// SIMATIC STEP 7 (V5.x) project LOCO#1ON_BOARD_PLC(TATA)
// CPU: CPU 315-2 DP
// station: P_ADR_BUS
// station: Hardware
// station: OB_PLC_QL--1
// program: S7 Program(1)

SYMBOL_TABLE
"RDREC"	SFB 52	SFB 52	// Read a Process Data Record
"WRREC"	SFB 53	SFB 53	// Write a Process Data Record
"RD_SINFO"	SFC 6	SFC 6	// Read OB Start Information
"BLKMOV"	SFC 20	SFC 20	// Copy Variables
"FILL"	SFC 21	SFC 21	// Initialize a Memory Area
"RDSYSST"	SFC 51	SFC 51	// Read a System Status List or Partial List
"WR_REC"	SFC 58	SFC 58	// Write Data Record
"RD_REC"	SFC 59	SFC 59	// Read a Data Record
END_SYMBOL_TABLE

// FB 7: know-how protected block, not included

// FB 8: know-how protected block, not included

// FC 1: know-how protected block, not included

// FC 2: know-how protected block, not included

// FC 3: know-how protected block, not included

// FC 4: know-how protected block, not included

FUNCTION FC 10 : VOID
VERSION : 0.1
BEGIN
// (block stored without names or comments; labels and parameter names are numbered)
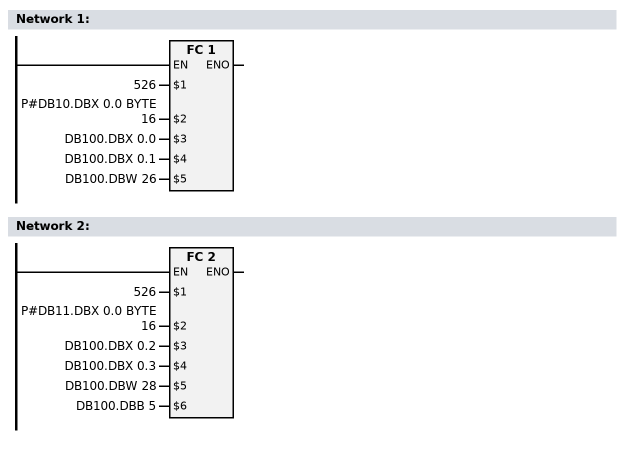
NETWORK
TITLE =
      CALL  FC 1 (
           $1                       := 526,
           $2                       := P#DB10.DBX 0.0 BYTE 16,
           $3                       := DB100.DBX 0.0,
           $4                       := DB100.DBX 0.1,
           $5                       := DB100.DBW 26);
      NOP   0;
NETWORK
TITLE =
      CALL  FC 2 (
           $1                       := 526,
           $2                       := P#DB11.DBX 0.0 BYTE 16,
           $3                       := DB100.DBX 0.2,
           $4                       := DB100.DBX 0.3,
           $5                       := DB100.DBW 28,
           $6                       := DB100.DBB 5);
      NOP   0;
END_FUNCTION

FUNCTION FC 14 : VOID
VERSION : 0.1
BEGIN
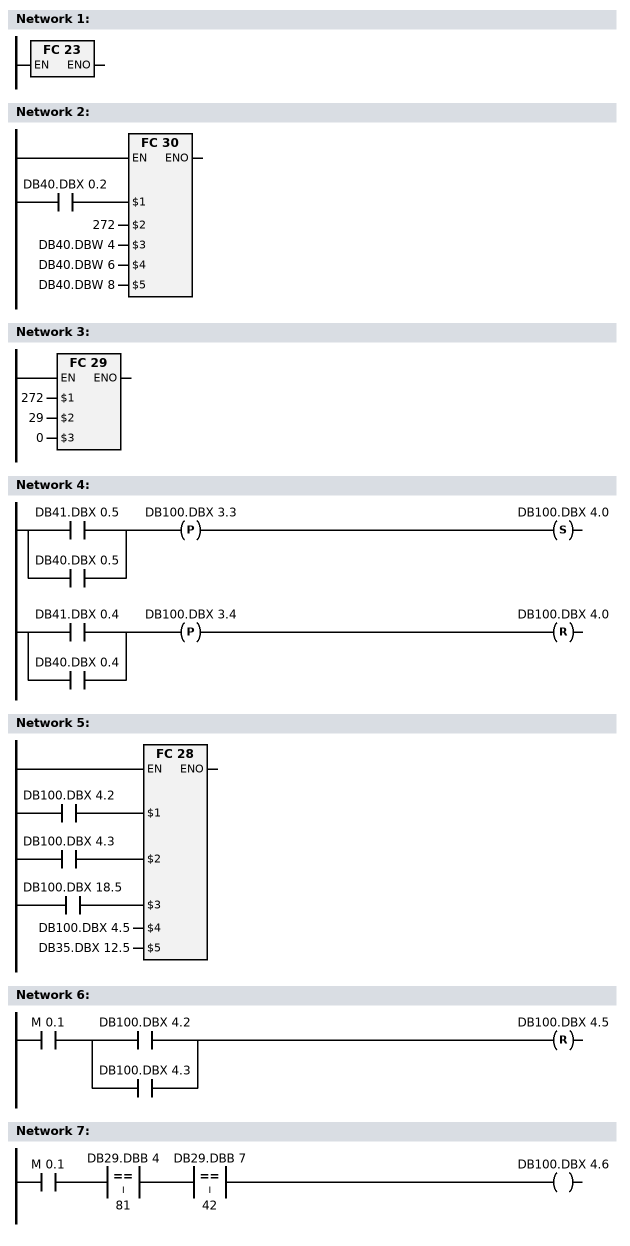
NETWORK
TITLE =
      CALL  FC 23;
      NOP   0;
NETWORK
TITLE =
      A     DB40.DBX 0.2;
      =     L 0.0;
      BLD   103;
      CALL  FC 30 (
           $1                       := L 0.0,
           $2                       := 272,
           $3                       := DB40.DBW 4,
           $4                       := DB40.DBW 6,
           $5                       := DB40.DBW 8);
      NOP   0;
NETWORK
TITLE =
      CALL  FC 29 (
           $1                       := 272,
           $2                       := 29,
           $3                       := 0);
      NOP   0;
NETWORK
TITLE =
      A(;
      O     DB41.DBX 0.5;
      O     DB40.DBX 0.5;
      );
      FP    DB100.DBX 3.3;
      S     DB100.DBX 4.0;
      A(;
      O     DB41.DBX 0.4;
      O     DB40.DBX 0.4;
      );
      FP    DB100.DBX 3.4;
      R     DB100.DBX 4.0;
      NOP   0;
NETWORK
TITLE =
      A     DB100.DBX 4.2;
      =     L 0.0;
      BLD   103;
      A     DB100.DBX 4.3;
      =     L 0.1;
      BLD   103;
      A     DB100.DBX 18.5;
      =     L 0.2;
      BLD   103;
      CALL  FC 28 (
           $1                       := L 0.0,
           $2                       := L 0.1,
           $3                       := L 0.2,
           $4                       := DB100.DBX 4.5,
           $5                       := DB35.DBX 12.5);
      NOP   0;
NETWORK
TITLE =
      A     M 0.1;
      A(;
      O     DB100.DBX 4.2;
      O     DB100.DBX 4.3;
      );
      R     DB100.DBX 4.5;
NETWORK
TITLE =
      A     M 0.1;
      A(;
      L     DB29.DBB 4;
      L     81;
      ==I;
      );
      A(;
      L     DB29.DBB 7;
      L     42;
      ==I;
      );
      =     DB100.DBX 4.6;
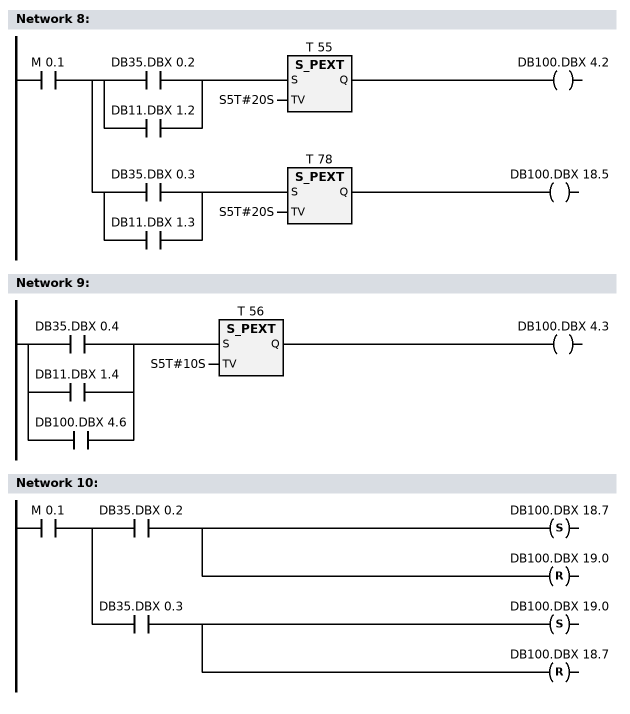
NETWORK
TITLE =
      A     M 0.1;
      =     L 0.0;
      A     L 0.0;
      A(;
      O     DB35.DBX 0.2;
      O     DB11.DBX 1.2;
      );
      L     S5T#20S;
      SE    T 55;
      NOP   0;
      NOP   0;
      NOP   0;
      A     T 55;
      =     DB100.DBX 4.2;
      A     L 0.0;
      A(;
      O     DB35.DBX 0.3;
      O     DB11.DBX 1.3;
      );
      L     S5T#20S;
      SE    T 78;
      NOP   0;
      NOP   0;
      NOP   0;
      A     T 78;
      =     DB100.DBX 18.5;
NETWORK
TITLE =
      A(;
      O     DB35.DBX 0.4;
      O     DB11.DBX 1.4;
      O     DB100.DBX 4.6;
      );
      L     S5T#10S;
      SE    T 56;
      NOP   0;
      NOP   0;
      NOP   0;
      A     T 56;
      =     DB100.DBX 4.3;
NETWORK
TITLE =
      A     M 0.1;
      =     L 0.0;
      A     L 0.0;
      A     DB35.DBX 0.2;
      S     DB100.DBX 18.7;
      R     DB100.DBX 19.0;
      A     L 0.0;
      A     DB35.DBX 0.3;
      S     DB100.DBX 19.0;
      R     DB100.DBX 18.7;
END_FUNCTION

FUNCTION FC 16 : VOID
VERSION : 0.1
BEGIN
// (block stored without names or comments; labels and parameter names are numbered)
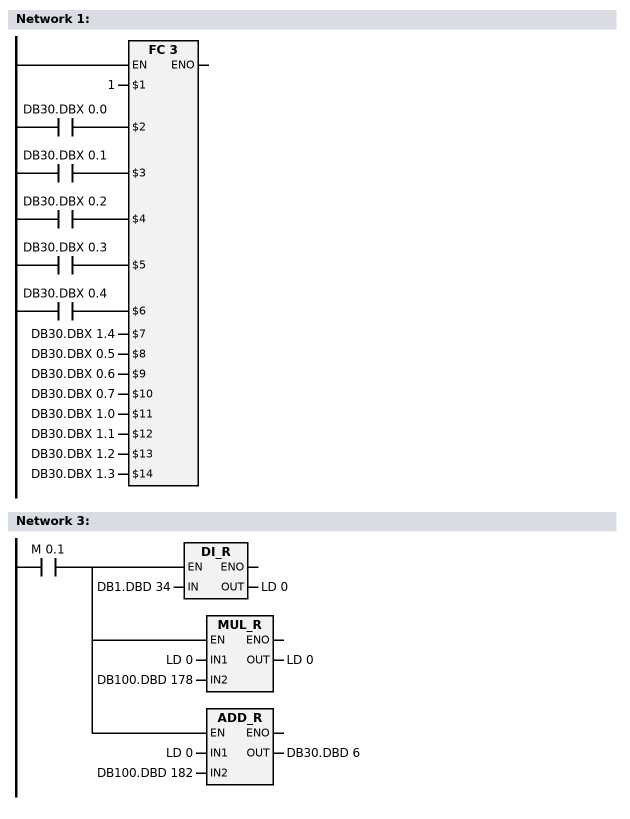
NETWORK
TITLE =
      A     DB30.DBX 0.0;
      =     L 4.0;
      BLD   103;
      A     DB30.DBX 0.1;
      =     L 4.1;
      BLD   103;
      A     DB30.DBX 0.2;
      =     L 4.2;
      BLD   103;
      A     DB30.DBX 0.3;
      =     L 4.3;
      BLD   103;
      A     DB30.DBX 0.4;
      =     L 4.4;
      BLD   103;
      CALL  FC 3 (
           $1                       := 1,
           $2                       := L 4.0,
           $3                       := L 4.1,
           $4                       := L 4.2,
           $5                       := L 4.3,
           $6                       := L 4.4,
           $7                       := DB30.DBX 1.4,
           $8                       := DB30.DBX 0.5,
           $9                       := DB30.DBX 0.6,
           $10                      := DB30.DBX 0.7,
           $11                      := DB30.DBX 1.0,
           $12                      := DB30.DBX 1.1,
           $13                      := DB30.DBX 1.2,
           $14                      := DB30.DBX 1.3);
      NOP   0;
NETWORK
TITLE =
NETWORK
TITLE =
      A     M 0.1;
      =     L 4.0;
      A     L 4.0;
      JNB   M001;
      L     DB1.DBD 34;
      DTR;
      T     LD 0;
M001: NOP   0;
      A     L 4.0;
      JNB   M002;
      L     LD 0;
      L     DB100.DBD 178;
      *R;
      T     LD 0;
M002: NOP   0;
      A     L 4.0;
      JNB   M003;
      L     LD 0;
      L     DB100.DBD 182;
      +R;
      T     DB30.DBD 6;
M003: NOP   0;
END_FUNCTION

FUNCTION FC 19 : VOID
VERSION : 0.1
BEGIN
// (block stored without names or comments; labels and parameter names are numbered)
NETWORK
TITLE =
      A     DB100.DBX 0.4;
      =     L 0.0;
      BLD   103;
      CALL  FC 31 (
           $1                       := L 0.0,
           $2                       := 288,
           $3                       := DB100.DBW 112,
           $4                       := P#M 45.0,
           $5                       := P#M 47.0,
           $6                       := DB31.DBX 2.0,
           $7                       := DB31.DBX 2.1,
           $8                       := DB31.DBX 2.2,
           $9                       := DB31.DBX 6.0,
           $10                      := DB31.DBX 2.3);
      NOP   0;
NETWORK
TITLE =
      L     MW 45;
      T     DB31.DBW 0;
      L     MW 47;
      T     DB31.DBW 4;
END_FUNCTION

FUNCTION FC 20 : VOID
VERSION : 0.1
BEGIN
// (block stored without names or comments; labels and parameter names are numbered)
NETWORK
TITLE =
      A     M 0.1;
      A(;
      L     DB21.DBW 46;
      L     1;
      ==I;
      );
      A(;
      L     DB21.DBB 50;
      L     'P';
      ==I;
      );
      JNB   M001;
      L     DB21.DBW 24;
      T     DB35.DBW 278;
M001: NOP   0;
NETWORK
TITLE =
      A     M 0.1;
      A(;
      L     DB21.DBW 46;
      L     1;
      ==I;
      );
      A(;
      L     DB21.DBB 50;
      L     'C';
      ==I;
      );
      A(;
      L     DB21.DBW 74;
      L     2;
      ==I;
      );
      A(;
      L     DB21.DBB 78;
      L     'P';
      ==I;
      );
      JNB   M002;
      L     DB21.DBW 52;
      T     DB35.DBW 278;
M002: NOP   0;
NETWORK
TITLE =
      A     M 0.1;
      A(;
      L     DB21.DBW 46;
      L     1;
      ==I;
      );
      A(;
      L     DB21.DBB 50;
      L     'C';
      ==I;
      );
      A(;
      L     DB21.DBW 74;
      L     2;
      ==I;
      );
      A(;
      L     DB21.DBB 78;
      L     'C';
      ==I;
      );
      A(;
      L     DB21.DBW 102;
      L     3;
      ==I;
      );
      A(;
      L     DB21.DBB 106;
      L     'P';
      ==I;
      );
      JNB   M003;
      L     DB21.DBW 80;
      T     DB35.DBW 278;
M003: NOP   0;
NETWORK
TITLE =
      A     M 0.1;
      A(;
      L     DB21.DBW 46;
      L     1;
      ==I;
      );
      A(;
      L     DB21.DBB 50;
      L     'C';
      ==I;
      );
      A(;
      L     DB21.DBW 74;
      L     2;
      ==I;
      );
      A(;
      L     DB21.DBB 78;
      L     'C';
      ==I;
      );
      A(;
      L     DB21.DBW 102;
      L     3;
      ==I;
      );
      A(;
      L     DB21.DBB 106;
      L     'C';
      ==I;
      );
      A(;
      L     DB21.DBW 130;
      L     4;
      ==I;
      );
      A(;
      L     DB21.DBB 134;
      L     'P';
      ==I;
      );
      JNB   M004;
      L     DB21.DBW 108;
      T     DB35.DBW 278;
M004: NOP   0;
NETWORK
TITLE =
      A     M 0.1;
      A(;
      L     DB21.DBW 46;
      L     1;
      ==I;
      );
      A(;
      L     DB21.DBB 50;
      L     'C';
      ==I;
      );
      =     L 0.0;
      A     L 0.0;
      JNB   M005;
      L     DB21.DBW 24;
      T     DB35.DBW 280;
M005: NOP   0;
      A     L 0.0;
      JNB   M006;
      L     DB21.DBB 50;
      T     DB35.DBB 284;
M006: NOP   0;
END_FUNCTION

FUNCTION FC 21 : VOID
VERSION : 0.1
BEGIN
// (block stored without names or comments; labels and parameter names are numbered)
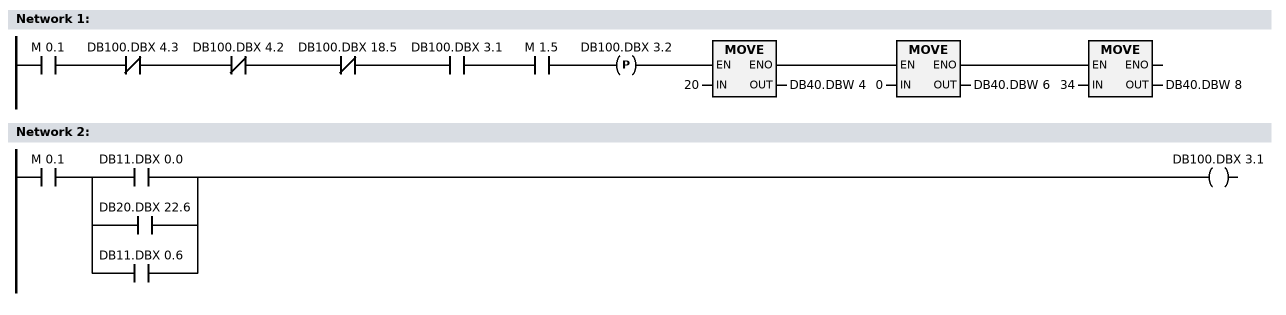
NETWORK
TITLE =
      A(;
      A(;
      A     M 0.1;
      AN    DB100.DBX 4.3;
      AN    DB100.DBX 4.2;
      AN    DB100.DBX 18.5;
      A     DB100.DBX 3.1;
      A     M 1.5;
      FP    DB100.DBX 3.2;
      JNB   M001;
      L     20;
      T     DB40.DBW 4;
      SET;
      SAVE;
      CLR;
M001: A     BR;
      );
      JNB   M002;
      L     0;
      T     DB40.DBW 6;
      SET;
      SAVE;
      CLR;
M002: A     BR;
      );
      JNB   M003;
      L     34;
      T     DB40.DBW 8;
M003: NOP   0;
NETWORK
TITLE =
      A     M 0.1;
      A(;
      O     DB11.DBX 0.0;
      O     DB20.DBX 22.6;
      O     DB11.DBX 0.6;
      );
      =     DB100.DBX 3.1;
END_FUNCTION

FUNCTION FC 22 : VOID
VERSION : 0.1
BEGIN
// (block stored without names or comments; labels and parameter names are numbered)
NETWORK
TITLE =
      A     DB41.DBX 0.4;
      A(;
      L     DB29.DBB 8;
      L     B#16#3;
      ==I;
      );
      A(;
      L     DB29.DBB 11;
      L     32;
      ==I;
      );
      =     DB100.DBX 15.1;
      A     DB100.DBX 15.1;
      FP    DB100.DBX 15.7;
      JNB   M001;
      CALL  "FILL" (
           BVAL                     := P#DB29.DBX 0.0 BYTE 30,
           RET_VAL                  := DB100.DBW 122,
           BLK                      := P#DB17.DBX 0.0 BYTE 30);
M001: NOP   0;
NETWORK
TITLE =
      A     DB41.DBX 0.4;
      A(;
      L     DB29.DBB 8;
      L     B#16#2;
      ==I;
      );
      A(;
      L     DB29.DBB 11;
      L     38;
      ==I;
      );
      =     DB100.DBX 15.0;
      A     DB100.DBX 15.0;
      FP    DB100.DBX 15.5;
      JNB   M002;
      CALL  "FILL" (
           BVAL                     := P#DB29.DBX 0.0 BYTE 34,
           RET_VAL                  := DB100.DBW 120,
           BLK                      := P#DB19.DBX 0.0 BYTE 34);
M002: NOP   0;
NETWORK
TITLE =
      A     DB41.DBX 0.4;
      A(;
      L     DB29.DBB 8;
      L     B#16#4;
      ==I;
      );
      A(;
      L     DB29.DBB 11;
      L     30;
      ==I;
      );
      =     DB100.DBX 15.2;
      A     DB100.DBX 15.2;
      FP    DB100.DBX 15.6;
      JNB   M003;
      CALL  "FILL" (
           BVAL                     := P#DB29.DBX 0.0 BYTE 30,
           RET_VAL                  := DB100.DBW 124,
           BLK                      := P#DB18.DBX 0.0 BYTE 30);
M003: NOP   0;
NETWORK
TITLE =
      A     DB41.DBX 0.4;
      A(;
      L     DB29.DBB 8;
      L     B#16#10;
      ==I;
      );
      A(;
      L     DB29.DBB 11;
      L     167;
      ==I;
      );
      =     DB100.DBX 15.4;
      A     DB100.DBX 15.4;
      FP    DB100.DBX 16.0;
      JNB   M004;
      CALL  "FILL" (
           BVAL                     := P#DB29.DBX 0.0 BYTE 167,
           RET_VAL                  := DB100.DBW 128,
           BLK                      := P#DB21.DBX 0.0 BYTE 167);
M004: NOP   0;
END_FUNCTION

FUNCTION FC 23 : VOID
VERSION : 0.1
BEGIN
// (block stored without names or comments; labels and parameter names are numbered)
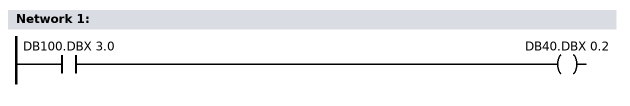
NETWORK
TITLE =
      A     DB100.DBX 3.0;
      =     DB40.DBX 0.2;
END_FUNCTION

FUNCTION FC 24 : VOID
VERSION : 0.1
BEGIN
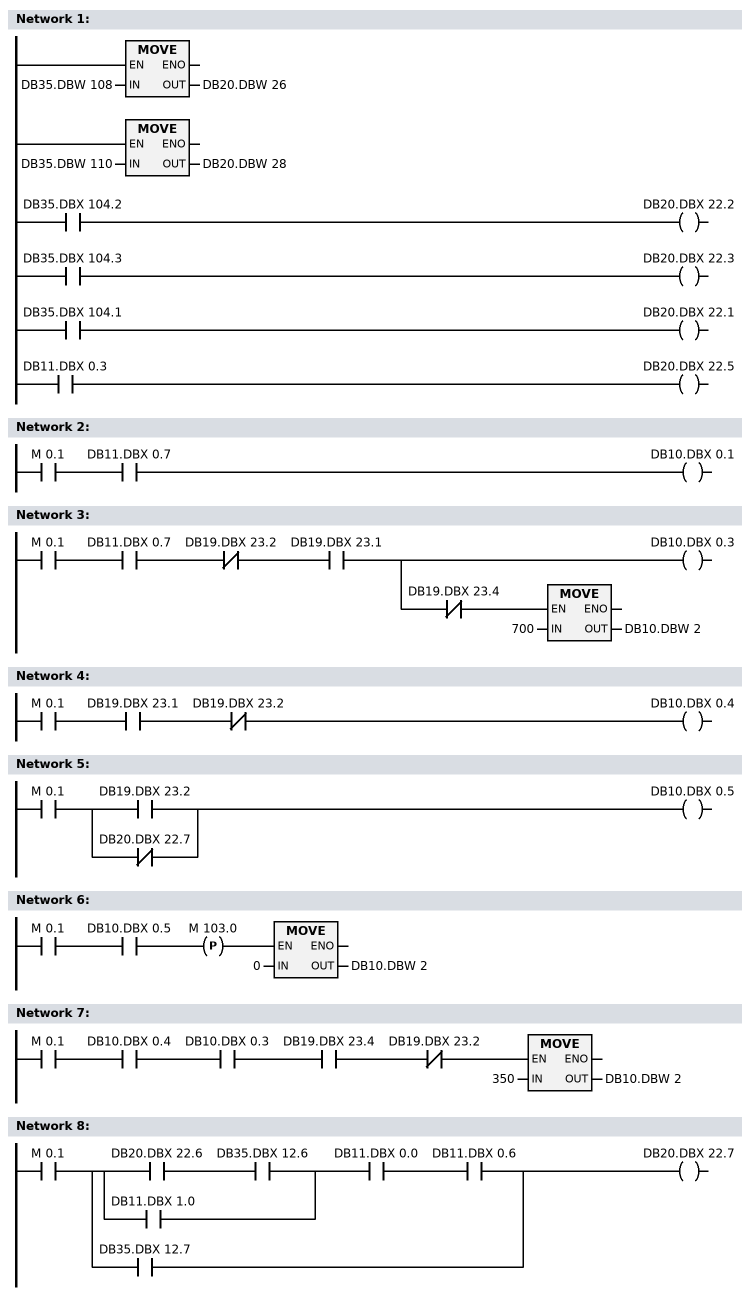
NETWORK
TITLE =
      L     DB35.DBW 108;
      T     DB20.DBW 26;
      L     DB35.DBW 110;
      T     DB20.DBW 28;
      A     DB35.DBX 104.2;
      =     DB20.DBX 22.2;
      A     DB35.DBX 104.3;
      =     DB20.DBX 22.3;
      A     DB35.DBX 104.1;
      =     DB20.DBX 22.1;
      A     DB11.DBX 0.3;
      =     DB20.DBX 22.5;
NETWORK
TITLE =
      A     M 0.1;
      A     DB11.DBX 0.7;
      =     DB10.DBX 0.1;
NETWORK
TITLE =
      A     M 0.1;
      A     DB11.DBX 0.7;
      AN    DB19.DBX 23.2;
      A     DB19.DBX 23.1;
      =     L 0.0;
      A     L 0.0;
      BLD   102;
      =     DB10.DBX 0.3;
      A     L 0.0;
      AN    DB19.DBX 23.4;
      JNB   _001;
      L     700;
      T     DB10.DBW 2;
_001: NOP   0;
NETWORK
TITLE =
      A     M 0.1;
      A     DB19.DBX 23.1;
      AN    DB19.DBX 23.2;
      =     DB10.DBX 0.4;
NETWORK
TITLE =
      A     M 0.1;
      A(;
      O     DB19.DBX 23.2;
      ON    DB20.DBX 22.7;
      );
      =     DB10.DBX 0.5;
NETWORK
TITLE =
      A     M 0.1;
      A     DB10.DBX 0.5;
      FP    M 103.0;
      JNB   _002;
      L     0;
      T     DB10.DBW 2;
_002: NOP   0;
NETWORK
TITLE =
      A     M 0.1;
      A     DB10.DBX 0.4;
      A     DB10.DBX 0.3;
      A     DB19.DBX 23.4;
      AN    DB19.DBX 23.2;
      JNB   _003;
      L     350;
      T     DB10.DBW 2;
_003: NOP   0;
NETWORK
TITLE =
      A     M 0.1;
      A(;
      A(;
      A     DB20.DBX 22.6;
      A     DB35.DBX 12.6;
      O     DB11.DBX 1.0;
      );
      A     DB11.DBX 0.0;
      A     DB11.DBX 0.6;
      O     DB35.DBX 12.7;
      );
      =     DB20.DBX 22.7;
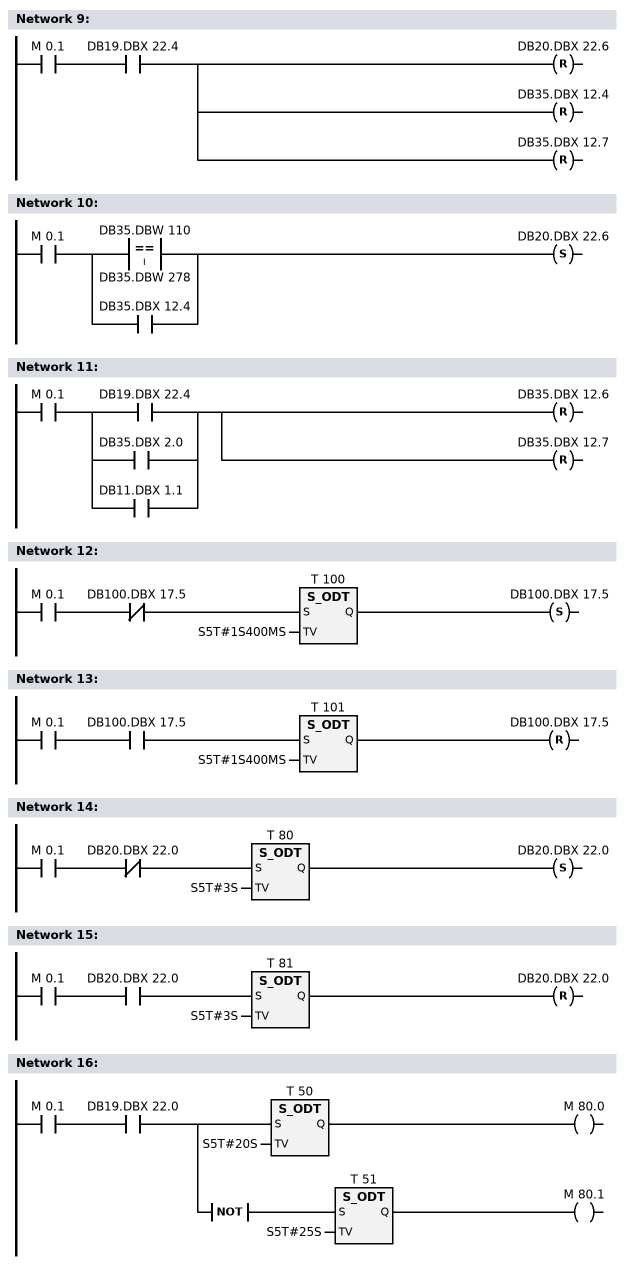
NETWORK
TITLE =
      A     M 0.1;
      A     DB19.DBX 22.4;
      R     DB20.DBX 22.6;
      R     DB35.DBX 12.4;
      R     DB35.DBX 12.7;
NETWORK
TITLE =
      A     M 0.1;
      A(;
      O(;
      L     DB35.DBW 110;
      L     DB35.DBW 278;
      ==I;
      );
      O     DB35.DBX 12.4;
      );
      S     DB20.DBX 22.6;
NETWORK
TITLE =
      A     M 0.1;
      A(;
      O     DB19.DBX 22.4;
      O     DB35.DBX 2.0;
      O     DB11.DBX 1.1;
      );
      R     DB35.DBX 12.6;
      R     DB35.DBX 12.7;
NETWORK
TITLE =
      A     M 0.1;
      AN    DB100.DBX 17.5;
      L     S5T#1S400MS;
      SD    T 100;
      NOP   0;
      NOP   0;
      NOP   0;
      A     T 100;
      S     DB100.DBX 17.5;
NETWORK
TITLE =
      A     M 0.1;
      A     DB100.DBX 17.5;
      L     S5T#1S400MS;
      SD    T 101;
      NOP   0;
      NOP   0;
      NOP   0;
      A     T 101;
      R     DB100.DBX 17.5;
NETWORK
TITLE =
      A     M 0.1;
      AN    DB20.DBX 22.0;
      L     S5T#3S;
      SD    T 80;
      NOP   0;
      NOP   0;
      NOP   0;
      A     T 80;
      S     DB20.DBX 22.0;
NETWORK
TITLE =
      A     M 0.1;
      A     DB20.DBX 22.0;
      L     S5T#3S;
      SD    T 81;
      NOP   0;
      NOP   0;
      NOP   0;
      A     T 81;
      R     DB20.DBX 22.0;
NETWORK
TITLE =
      A     M 0.1;
      A     DB19.DBX 22.0;
      =     L 0.0;
      A     L 0.0;
      L     S5T#20S;
      SD    T 50;
      NOP   0;
      NOP   0;
      NOP   0;
      A     T 50;
      =     M 80.0;
      A     L 0.0;
      NOT;
      L     S5T#25S;
      SD    T 51;
      NOP   0;
      NOP   0;
      NOP   0;
      A     T 51;
      =     M 80.1;
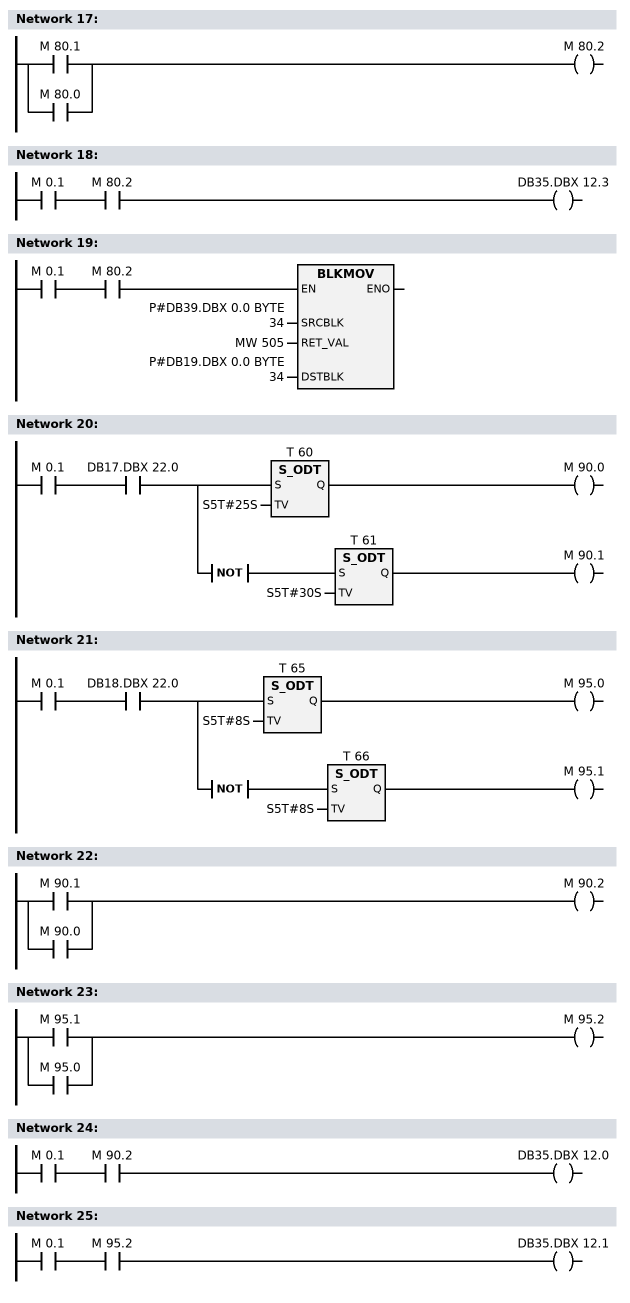
NETWORK
TITLE =
      O     M 80.1;
      O     M 80.0;
      =     M 80.2;
NETWORK
TITLE =
      A     M 0.1;
      A     M 80.2;
      =     DB35.DBX 12.3;
NETWORK
TITLE =
      A     M 0.1;
      A     M 80.2;
      JNB   _004;
      CALL  "BLKMOV" (
           SRCBLK                   := P#DB39.DBX 0.0 BYTE 34,
           RET_VAL                  := MW 505,
           DSTBLK                   := P#DB19.DBX 0.0 BYTE 34);
_004: NOP   0;
NETWORK
TITLE =
      A     M 0.1;
      A     DB17.DBX 22.0;
      =     L 0.0;
      A     L 0.0;
      L     S5T#25S;
      SD    T 60;
      NOP   0;
      NOP   0;
      NOP   0;
      A     T 60;
      =     M 90.0;
      A     L 0.0;
      NOT;
      L     S5T#30S;
      SD    T 61;
      NOP   0;
      NOP   0;
      NOP   0;
      A     T 61;
      =     M 90.1;
NETWORK
TITLE =
      A     M 0.1;
      A     DB18.DBX 22.0;
      =     L 0.0;
      A     L 0.0;
      L     S5T#8S;
      SD    T 65;
      NOP   0;
      NOP   0;
      NOP   0;
      A     T 65;
      =     M 95.0;
      A     L 0.0;
      NOT;
      L     S5T#8S;
      SD    T 66;
      NOP   0;
      NOP   0;
      NOP   0;
      A     T 66;
      =     M 95.1;
NETWORK
TITLE =
      O     M 90.1;
      O     M 90.0;
      =     M 90.2;
NETWORK
TITLE =
      O     M 95.1;
      O     M 95.0;
      =     M 95.2;
NETWORK
TITLE =
      A     M 0.1;
      A     M 90.2;
      =     DB35.DBX 12.0;
NETWORK
TITLE =
      A     M 0.1;
      A     M 95.2;
      =     DB35.DBX 12.1;
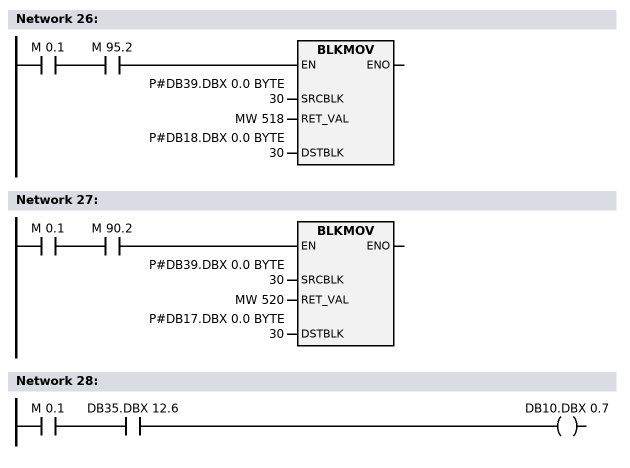
NETWORK
TITLE =
      A     M 0.1;
      A     M 95.2;
      JNB   _005;
      CALL  "BLKMOV" (
           SRCBLK                   := P#DB39.DBX 0.0 BYTE 30,
           RET_VAL                  := MW 518,
           DSTBLK                   := P#DB18.DBX 0.0 BYTE 30);
_005: NOP   0;
NETWORK
TITLE =
      A     M 0.1;
      A     M 90.2;
      JNB   _006;
      CALL  "BLKMOV" (
           SRCBLK                   := P#DB39.DBX 0.0 BYTE 30,
           RET_VAL                  := MW 520,
           DSTBLK                   := P#DB17.DBX 0.0 BYTE 30);
_006: NOP   0;
NETWORK
TITLE =
      A     M 0.1;
      A     DB35.DBX 12.6;
      =     DB10.DBX 0.7;
END_FUNCTION

FUNCTION FC 26 : VOID
VERSION : 0.1
BEGIN
// (block stored without names or comments; labels and parameter names are numbered)
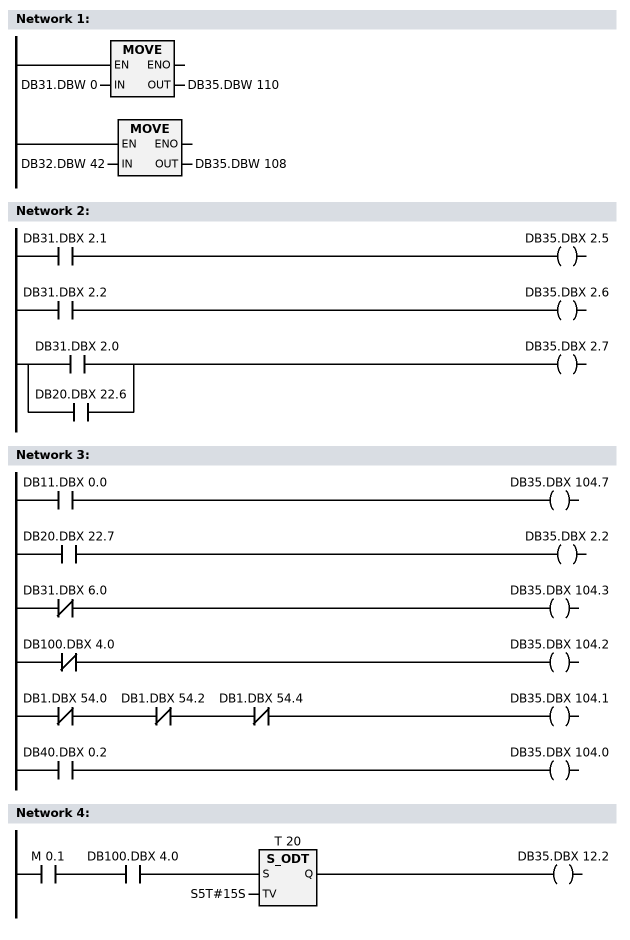
NETWORK
TITLE =
      L     DB31.DBW 0;
      T     DB35.DBW 110;
      L     DB32.DBW 42;
      T     DB35.DBW 108;
NETWORK
TITLE =
      A     DB31.DBX 2.1;
      =     DB35.DBX 2.5;
      A     DB31.DBX 2.2;
      =     DB35.DBX 2.6;
      O     DB31.DBX 2.0;
      O     DB20.DBX 22.6;
      =     DB35.DBX 2.7;
NETWORK
TITLE =
      A     DB11.DBX 0.0;
      =     DB35.DBX 104.7;
      A     DB20.DBX 22.7;
      =     DB35.DBX 2.2;
      AN    DB31.DBX 6.0;
      =     DB35.DBX 104.3;
      AN    DB100.DBX 4.0;
      =     DB35.DBX 104.2;
      AN    DB1.DBX 54.0;
      AN    DB1.DBX 54.2;
      AN    DB1.DBX 54.4;
      =     DB35.DBX 104.1;
      A     DB40.DBX 0.2;
      =     DB35.DBX 104.0;
NETWORK
TITLE =
      A     M 0.1;
      A     DB100.DBX 4.0;
      L     S5T#15S;
      SD    T 20;
      NOP   0;
      NOP   0;
      NOP   0;
      A     T 20;
      =     DB35.DBX 12.2;
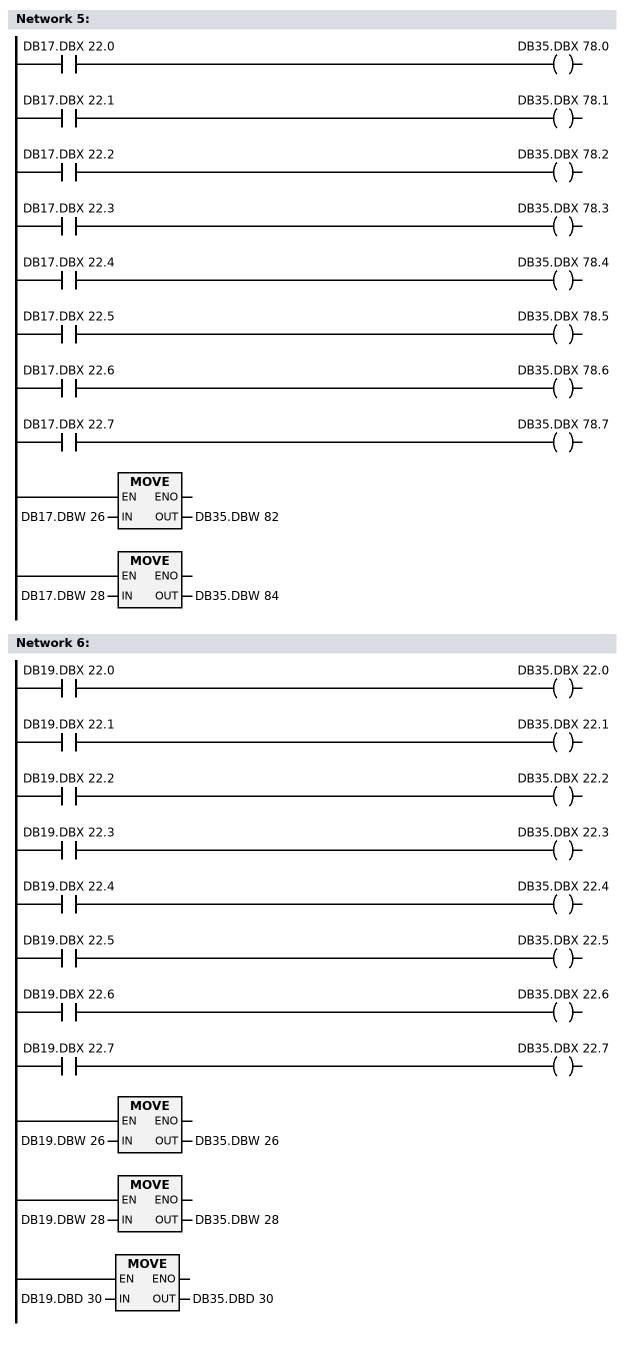
NETWORK
TITLE =
      A     DB17.DBX 22.0;
      =     DB35.DBX 78.0;
      A     DB17.DBX 22.1;
      =     DB35.DBX 78.1;
      A     DB17.DBX 22.2;
      =     DB35.DBX 78.2;
      A     DB17.DBX 22.3;
      =     DB35.DBX 78.3;
      A     DB17.DBX 22.4;
      =     DB35.DBX 78.4;
      A     DB17.DBX 22.5;
      =     DB35.DBX 78.5;
      A     DB17.DBX 22.6;
      =     DB35.DBX 78.6;
      A     DB17.DBX 22.7;
      =     DB35.DBX 78.7;
      L     DB17.DBW 26;
      T     DB35.DBW 82;
      L     DB17.DBW 28;
      T     DB35.DBW 84;
NETWORK
TITLE =
      A     DB19.DBX 22.0;
      =     DB35.DBX 22.0;
      A     DB19.DBX 22.1;
      =     DB35.DBX 22.1;
      A     DB19.DBX 22.2;
      =     DB35.DBX 22.2;
      A     DB19.DBX 22.3;
      =     DB35.DBX 22.3;
      A     DB19.DBX 22.4;
      =     DB35.DBX 22.4;
      A     DB19.DBX 22.5;
      =     DB35.DBX 22.5;
      A     DB19.DBX 22.6;
      =     DB35.DBX 22.6;
      A     DB19.DBX 22.7;
      =     DB35.DBX 22.7;
      L     DB19.DBW 26;
      T     DB35.DBW 26;
      L     DB19.DBW 28;
      T     DB35.DBW 28;
      L     DB19.DBD 30;
      T     DB35.DBD 30;
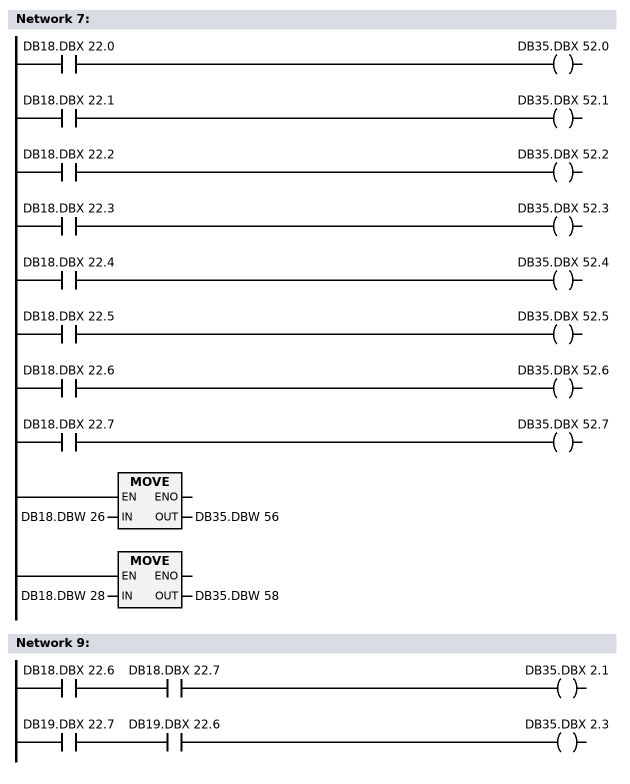
NETWORK
TITLE =
      A     DB18.DBX 22.0;
      =     DB35.DBX 52.0;
      A     DB18.DBX 22.1;
      =     DB35.DBX 52.1;
      A     DB18.DBX 22.2;
      =     DB35.DBX 52.2;
      A     DB18.DBX 22.3;
      =     DB35.DBX 52.3;
      A     DB18.DBX 22.4;
      =     DB35.DBX 52.4;
      A     DB18.DBX 22.5;
      =     DB35.DBX 52.5;
      A     DB18.DBX 22.6;
      =     DB35.DBX 52.6;
      A     DB18.DBX 22.7;
      =     DB35.DBX 52.7;
      L     DB18.DBW 26;
      T     DB35.DBW 56;
      L     DB18.DBW 28;
      T     DB35.DBW 58;
NETWORK
TITLE =
NETWORK
TITLE =
      A     DB18.DBX 22.6;
      A     DB18.DBX 22.7;
      =     DB35.DBX 2.1;
      A     DB19.DBX 22.7;
      A     DB19.DBX 22.6;
      =     DB35.DBX 2.3;
END_FUNCTION

FUNCTION FC 28 : VOID
VERSION : 0.1
BEGIN
// (block stored without names or comments; labels and parameter names are numbered)
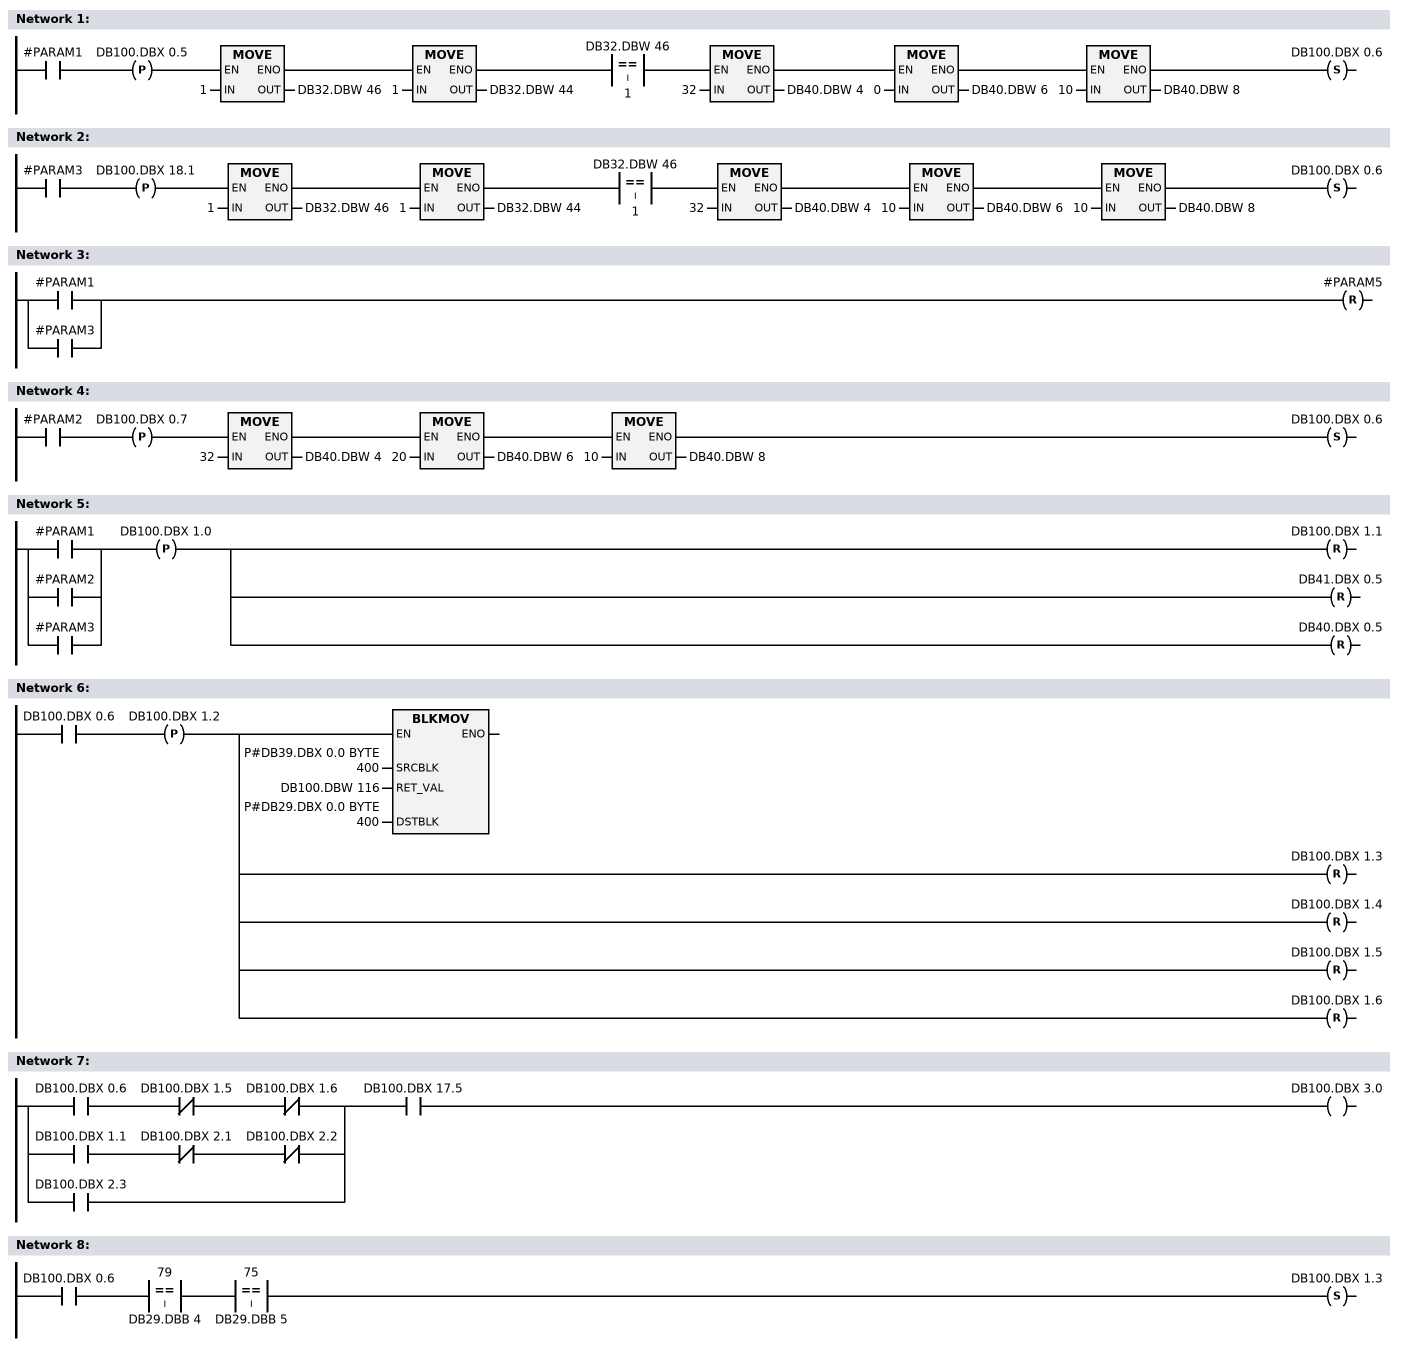
NETWORK
TITLE =
      A(;
      A(;
      A(;
      A(;
      A     #PARAM1;
      FP    DB100.DBX 0.5;
      JNB   M001;
      L     1;
      T     DB32.DBW 46;
      SET;
      SAVE;
      CLR;
M001: A     BR;
      );
      JNB   M002;
      L     1;
      T     DB32.DBW 44;
      SET;
      SAVE;
      CLR;
M002: A     BR;
      );
      A(;
      L     DB32.DBW 46;
      L     1;
      ==I;
      );
      JNB   M003;
      L     32;
      T     DB40.DBW 4;
      SET;
      SAVE;
      CLR;
M003: A     BR;
      );
      JNB   M004;
      L     0;
      T     DB40.DBW 6;
      SET;
      SAVE;
      CLR;
M004: A     BR;
      );
      JNB   M005;
      L     10;
      T     DB40.DBW 8;
      SET;
      SAVE;
      CLR;
M005: A     BR;
      S     DB100.DBX 0.6;
NETWORK
TITLE =
      A(;
      A(;
      A(;
      A(;
      A     #PARAM3;
      FP    DB100.DBX 18.1;
      JNB   M006;
      L     1;
      T     DB32.DBW 46;
      SET;
      SAVE;
      CLR;
M006: A     BR;
      );
      JNB   M007;
      L     1;
      T     DB32.DBW 44;
      SET;
      SAVE;
      CLR;
M007: A     BR;
      );
      A(;
      L     DB32.DBW 46;
      L     1;
      ==I;
      );
      JNB   M008;
      L     32;
      T     DB40.DBW 4;
      SET;
      SAVE;
      CLR;
M008: A     BR;
      );
      JNB   M009;
      L     10;
      T     DB40.DBW 6;
      SET;
      SAVE;
      CLR;
M009: A     BR;
      );
      JNB   M010;
      L     10;
      T     DB40.DBW 8;
      SET;
      SAVE;
      CLR;
M010: A     BR;
      S     DB100.DBX 0.6;
NETWORK
TITLE =
      O     #PARAM1;
      O     #PARAM3;
      R     #PARAM5;
NETWORK
TITLE =
      A(;
      A(;
      A     #PARAM2;
      FP    DB100.DBX 0.7;
      JNB   M011;
      L     32;
      T     DB40.DBW 4;
      SET;
      SAVE;
      CLR;
M011: A     BR;
      );
      JNB   M012;
      L     20;
      T     DB40.DBW 6;
      SET;
      SAVE;
      CLR;
M012: A     BR;
      );
      JNB   M013;
      L     10;
      T     DB40.DBW 8;
      SET;
      SAVE;
      CLR;
M013: A     BR;
      S     DB100.DBX 0.6;
NETWORK
TITLE =
      A(;
      O     #PARAM1;
      O     #PARAM2;
      O     #PARAM3;
      );
      FP    DB100.DBX 1.0;
      R     DB100.DBX 1.1;
      R     DB41.DBX 0.5;
      R     DB40.DBX 0.5;
NETWORK
TITLE =
      A     DB100.DBX 0.6;
      FP    DB100.DBX 1.2;
      =     L 0.0;
      A     L 0.0;
      JNB   M014;
      CALL  "BLKMOV" (
           SRCBLK                   := P#DB39.DBX 0.0 BYTE 400,
           RET_VAL                  := DB100.DBW 116,
           DSTBLK                   := P#DB29.DBX 0.0 BYTE 400);
M014: NOP   0;
      A     L 0.0;
      BLD   102;
      R     DB100.DBX 1.3;
      A     L 0.0;
      BLD   102;
      R     DB100.DBX 1.4;
      A     L 0.0;
      BLD   102;
      R     DB100.DBX 1.5;
      A     L 0.0;
      BLD   102;
      R     DB100.DBX 1.6;
NETWORK
TITLE =
      A(;
      A     DB100.DBX 0.6;
      AN    DB100.DBX 1.5;
      AN    DB100.DBX 1.6;
      O;
      A     DB100.DBX 1.1;
      AN    DB100.DBX 2.1;
      AN    DB100.DBX 2.2;
      O     DB100.DBX 2.3;
      );
      A     DB100.DBX 17.5;
      =     DB100.DBX 3.0;
NETWORK
TITLE =
      A     DB100.DBX 0.6;
      A(;
      L     79;
      L     DB29.DBB 4;
      ==I;
      );
      A(;
      L     75;
      L     DB29.DBB 5;
      ==I;
      );
      S     DB100.DBX 1.3;
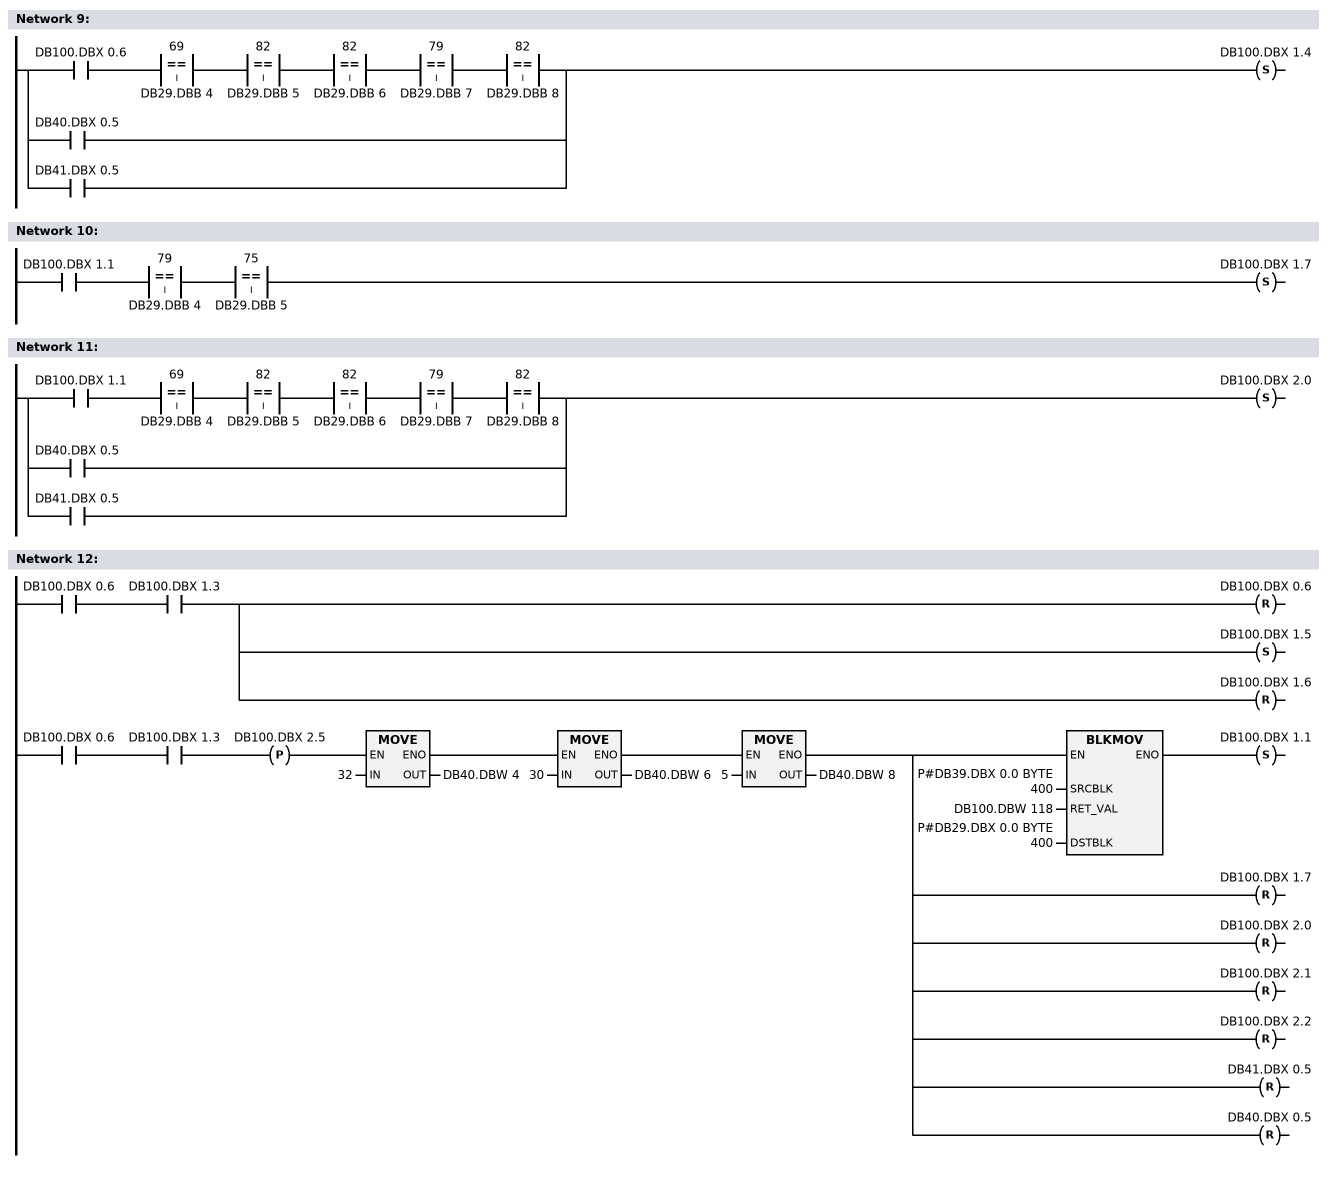
NETWORK
TITLE =
      A     DB100.DBX 0.6;
      A(;
      L     69;
      L     DB29.DBB 4;
      ==I;
      );
      A(;
      L     82;
      L     DB29.DBB 5;
      ==I;
      );
      A(;
      L     82;
      L     DB29.DBB 6;
      ==I;
      );
      A(;
      L     79;
      L     DB29.DBB 7;
      ==I;
      );
      A(;
      L     82;
      L     DB29.DBB 8;
      ==I;
      );
      O     DB40.DBX 0.5;
      O     DB41.DBX 0.5;
      S     DB100.DBX 1.4;
NETWORK
TITLE =
      A     DB100.DBX 1.1;
      A(;
      L     79;
      L     DB29.DBB 4;
      ==I;
      );
      A(;
      L     75;
      L     DB29.DBB 5;
      ==I;
      );
      S     DB100.DBX 1.7;
NETWORK
TITLE =
      A     DB100.DBX 1.1;
      A(;
      L     69;
      L     DB29.DBB 4;
      ==I;
      );
      A(;
      L     82;
      L     DB29.DBB 5;
      ==I;
      );
      A(;
      L     82;
      L     DB29.DBB 6;
      ==I;
      );
      A(;
      L     79;
      L     DB29.DBB 7;
      ==I;
      );
      A(;
      L     82;
      L     DB29.DBB 8;
      ==I;
      );
      O     DB40.DBX 0.5;
      O     DB41.DBX 0.5;
      S     DB100.DBX 2.0;
NETWORK
TITLE =
      A     DB100.DBX 0.6;
      A     DB100.DBX 1.3;
      =     L 0.0;
      A     L 0.0;
      BLD   102;
      R     DB100.DBX 0.6;
      A     L 0.0;
      BLD   102;
      S     DB100.DBX 1.5;
      A     L 0.0;
      BLD   102;
      R     DB100.DBX 1.6;
      A(;
      A(;
      A     L 0.0;
      FP    DB100.DBX 2.5;
      JNB   M015;
      L     32;
      T     DB40.DBW 4;
      SET;
      SAVE;
      CLR;
M015: A     BR;
      );
      JNB   M016;
      L     30;
      T     DB40.DBW 6;
      SET;
      SAVE;
      CLR;
M016: A     BR;
      );
      JNB   M017;
      L     5;
      T     DB40.DBW 8;
      SET;
      SAVE;
      CLR;
M017: A     BR;
      =     L 0.1;
      A     L 0.1;
      JNB   M018;
      CALL  "BLKMOV" (
           SRCBLK                   := P#DB39.DBX 0.0 BYTE 400,
           RET_VAL                  := DB100.DBW 118,
           DSTBLK                   := P#DB29.DBX 0.0 BYTE 400);
M018: A     BR;
      S     DB100.DBX 1.1;
      A     L 0.1;
      BLD   102;
      R     DB100.DBX 1.7;
      A     L 0.1;
      BLD   102;
      R     DB100.DBX 2.0;
      A     L 0.1;
      BLD   102;
      R     DB100.DBX 2.1;
      A     L 0.1;
      BLD   102;
      R     DB100.DBX 2.2;
      A     L 0.1;
      BLD   102;
      R     DB41.DBX 0.5;
      A     L 0.1;
      BLD   102;
      R     DB40.DBX 0.5;
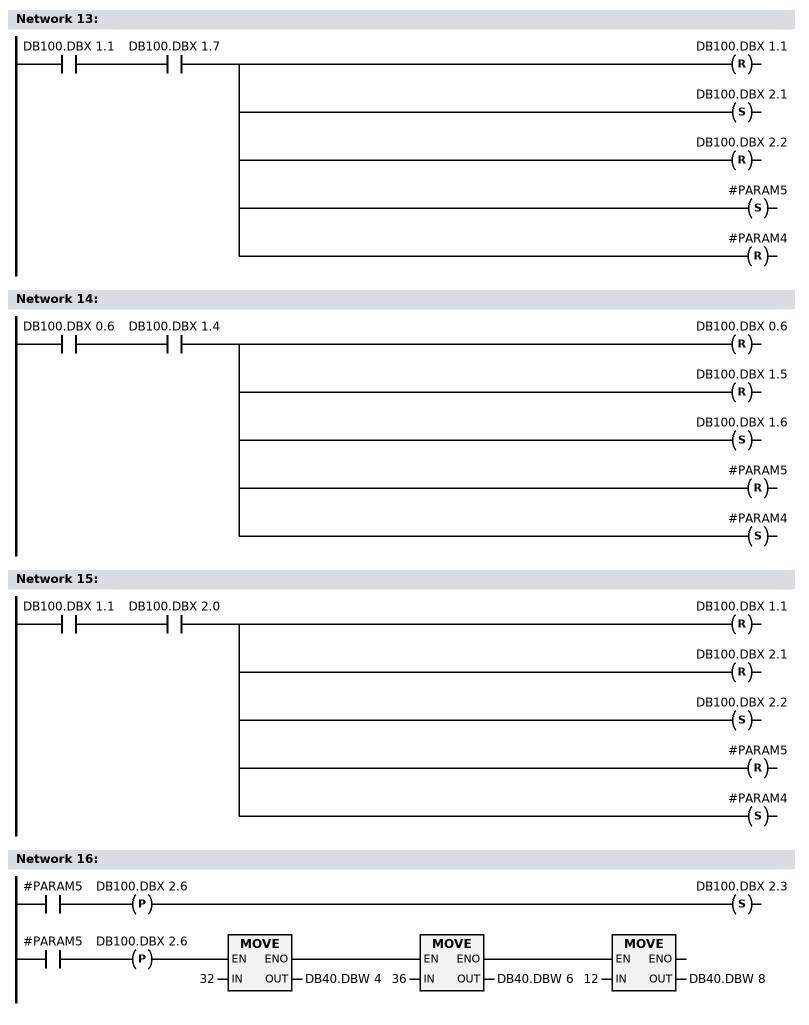
NETWORK
TITLE =
      A     DB100.DBX 1.1;
      A     DB100.DBX 1.7;
      R     DB100.DBX 1.1;
      S     DB100.DBX 2.1;
      R     DB100.DBX 2.2;
      S     #PARAM5;
      R     #PARAM4;
NETWORK
TITLE =
      A     DB100.DBX 0.6;
      A     DB100.DBX 1.4;
      R     DB100.DBX 0.6;
      R     DB100.DBX 1.5;
      S     DB100.DBX 1.6;
      R     #PARAM5;
      S     #PARAM4;
NETWORK
TITLE =
      A     DB100.DBX 1.1;
      A     DB100.DBX 2.0;
      R     DB100.DBX 1.1;
      R     DB100.DBX 2.1;
      S     DB100.DBX 2.2;
      R     #PARAM5;
      S     #PARAM4;
NETWORK
TITLE =
      A     #PARAM5;
      FP    DB100.DBX 2.6;
      =     L 0.0;
      A     L 0.0;
      BLD   102;
      S     DB100.DBX 2.3;
      A(;
      A(;
      A     L 0.0;
      JNB   M019;
      L     32;
      T     DB40.DBW 4;
      SET;
      SAVE;
      CLR;
M019: A     BR;
      );
      JNB   M020;
      L     36;
      T     DB40.DBW 6;
      SET;
      SAVE;
      CLR;
M020: A     BR;
      );
      JNB   M021;
      L     12;
      T     DB40.DBW 8;
M021: NOP   0;
NETWORK
TITLE =
NETWORK
TITLE =
NETWORK
TITLE =
      BE;
END_FUNCTION

FUNCTION FC 29 : VOID
VERSION : 0.1
BEGIN
// (block stored without names or comments; labels and parameter names are numbered)
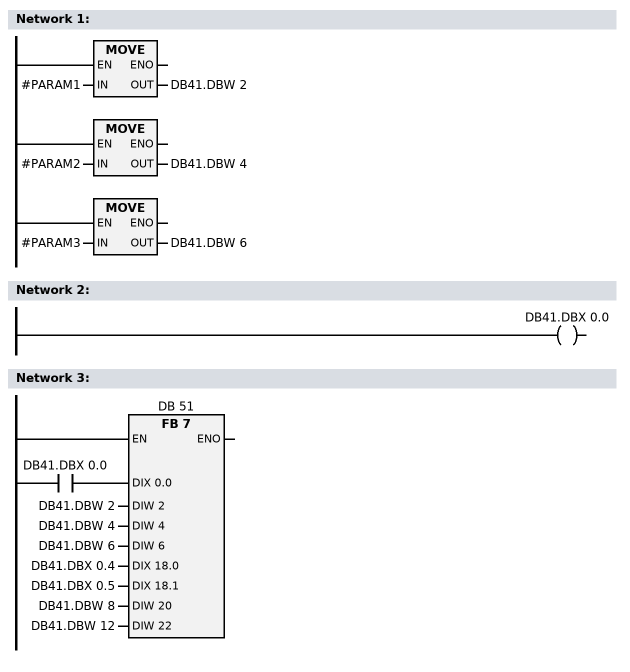
NETWORK
TITLE =
      L     #PARAM1;
      T     DB41.DBW 2;
      L     #PARAM2;
      T     DB41.DBW 4;
      L     #PARAM3;
      T     DB41.DBW 6;
NETWORK
TITLE =
      SET;
      =     DB41.DBX 0.0;
NETWORK
TITLE =
      A     DB41.DBX 0.0;
      =     L 0.0;
      BLD   103;
      CALL  FB 7 , DB 51 (
           DIX 0.0                  := L 0.0,
           DIW 2                    := DB41.DBW 2,
           DIW 4                    := DB41.DBW 4,
           DIW 6                    := DB41.DBW 6,
           DIX 18.0                 := DB41.DBX 0.4,
           DIX 18.1                 := DB41.DBX 0.5,
           DIW 20                   := DB41.DBW 8,
           DIW 22                   := DB41.DBW 12);
      NOP   0;
NETWORK
TITLE =
      AN    DB41.DBX 0.4;
      JC    M001;
      L     DB41.DBW 18;
      +     1;
      T     DB41.DBW 18;
      L     DB41.DBW 8;
      T     DB41.DBW 10;
      BE;
M001: AN    DB41.DBX 0.5;
      BEC;
      L     DB41.DBW 20;
      +     1;
      T     DB41.DBW 20;
      L     DB41.DBW 12;
      T     DB41.DBW 14;
      BE;
NETWORK
TITLE =
END_FUNCTION

FUNCTION FC 30 : VOID
VERSION : 0.1
BEGIN
// (block stored without names or comments; labels and parameter names are numbered)
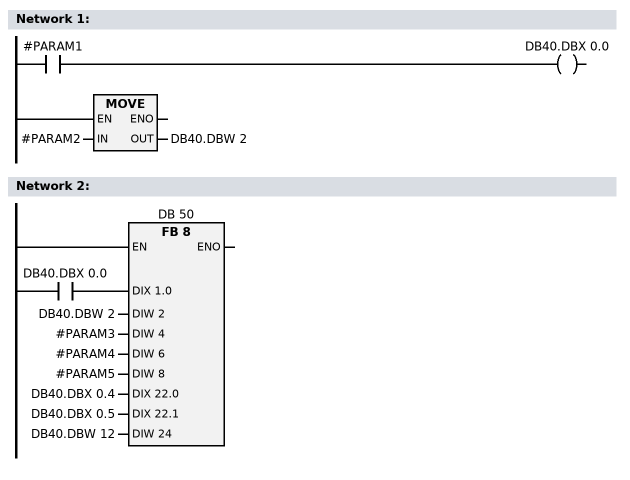
NETWORK
TITLE =
      A     #PARAM1;
      =     DB40.DBX 0.0;
      L     #PARAM2;
      T     DB40.DBW 2;
NETWORK
TITLE =
      A     DB40.DBX 0.0;
      =     L 0.0;
      BLD   103;
      CALL  FB 8 , DB 50 (
           DIX 1.0                  := L 0.0,
           DIW 2                    := DB40.DBW 2,
           DIW 4                    := #PARAM3,
           DIW 6                    := #PARAM4,
           DIW 8                    := #PARAM5,
           DIX 22.0                 := DB40.DBX 0.4,
           DIX 22.1                 := DB40.DBX 0.5,
           DIW 24                   := DB40.DBW 12);
      NOP   0;
NETWORK
TITLE =
      AN    DB40.DBX 0.4;
      JC    M001;
      L     DB40.DBW 16;
      +     1;
      T     DB40.DBW 16;
      NOP   0;
      NOP   0;
      NOP   0;
      BE;
M001: AN    DB40.DBX 0.5;
      BEC;
      L     DB40.DBW 18;
      +     1;
      T     DB40.DBW 18;
      L     DB40.DBW 12;
      T     DB40.DBW 14;
      NOP   0;
      NOP   0;
      NOP   0;
      BE;
NETWORK
TITLE =
END_FUNCTION

FUNCTION FC 31 : VOID
VERSION : 0.1
BEGIN
// (block stored without names or comments; labels and parameter names are numbered)
NETWORK
TITLE =
      SET;
      =     #PARAM1;
NETWORK
TITLE =
      A     #PARAM1;
      =     L 4.0;
      BLD   103;
      CALL  FB 7 , DB 80 (
           DIX 0.0                  := L 4.0,
           DIW 2                    := #PARAM2,
           DIW 4                    := 31,
           DIW 6                    := 50,
           DIX 18.0                 := DB31.DBX 8.0,
           DIX 18.1                 := DB31.DBX 8.1,
           DIW 20                   := DB31.DBW 10,
           DIW 22                   := DB31.DBW 12);
      NOP   0;
NETWORK
TITLE =
      A     #PARAM1;
      A     DB31.DBX 8.0;
      AN    DB31.DBX 8.1;
      A(;
      L     DB31.DBW 12;
      L     0;
      ==I;
      );
      =     DB31.DBX 14.0;
NETWORK
TITLE =
      A     #PARAM1;
      A     DB31.DBX 14.0;
      A(;
      L     DB31.DBB 50;
      L     B#16#AA;
      ==I;
      );
      A(;
      O(;
      L     DB31.DBB 51;
      L     B#16#1;
      ==I;
      );
      O(;
      L     DB31.DBB 51;
      L     B#16#2;
      ==I;
      );
      );
      A(;
      L     DB31.DBB 59;
      L     B#16#20;
      ==I;
      );
      A(;
      L     DB31.DBB 60;
      L     B#16#D;
      ==I;
      );
      A(;
      L     DB31.DBB 61;
      L     B#16#A;
      ==I;
      );
      =     DB31.DBX 14.1;
NETWORK
TITLE =
      A     M 1.5;
      CU    C 127;
      BLD   101;
      NOP   0;
      NOP   0;
      A     DB31.DBX 14.1;
      R     C 127;
      L     C 127;
      T     LW 0;
      NOP   0;
      NOP   0;
NETWORK
TITLE =
      L     LW 0;
      L     3;
      >=I;
      =     DB31.DBX 14.2;
NETWORK
TITLE =
      A     DB31.DBX 14.2;
      =     #PARAM9;
NETWORK
TITLE =
      AN    DB31.DBX 14.2;
      A(;
      O(;
      L     DB31.DBB 51;
      L     B#16#1;
      ==I;
      );
      O(;
      L     DB31.DBB 51;
      L     B#16#2;
      ==I;
      );
      );
      =     L 2.0;
      A     L 2.0;
      A(;
      L     DB31.DBB 52;
      L     B#16#3;
      ==I;
      );
      =     #PARAM6;
      A     L 2.0;
      A(;
      L     DB31.DBB 52;
      L     B#16#2;
      ==I;
      );
      =     #PARAM8;
      A     L 2.0;
      A(;
      L     DB31.DBB 52;
      L     B#16#1;
      ==I;
      );
      =     #PARAM7;
NETWORK
TITLE =
      A     DB31.DBX 14.0;
      A     DB31.DBX 14.1;
      AN    DB31.DBX 14.2;
      A(;
      L     DB31.DBB 51;
      L     B#16#1;
      ==I;
      );
      A(;
      L     DB31.DBB 52;
      L     B#16#3;
      ==I;
      );
      JNB   M001;
      L     DB31.DBB 53;
      L     100;
      +I;
      T     #PARAM4;
M001: NOP   0;
NETWORK
TITLE =
      A(;
      L     #PARAM3;
      L     2;
      ==I;
      );
      A(;
      L     DB31.DBB 53;
      L     0;
      >=I;
      );
      A(;
      L     DB31.DBB 53;
      L     69;
      <=I;
      );
      O;
      A(;
      L     #PARAM3;
      L     1;
      ==I;
      );
      A(;
      L     DB31.DBB 53;
      L     100;
      >=I;
      );
      A(;
      L     DB31.DBB 53;
      L     169;
      <=I;
      );
      =     #PARAM10;
NETWORK
TITLE =
      L     DB31.DBB 58;
      T     #PARAM5;
NETWORK
TITLE =
      A     DB31.DBX 8.0;
      JCN   M002;
      L     DB31.DBW 18;
      +     1;
      T     DB31.DBW 18;
      L     DB31.DBW 10;
      T     DB31.DBW 16;
      JU    M004;
M002: A     DB31.DBX 8.1;
      JCN   M003;
      L     DB31.DBW 20;
      +     1;
      T     DB31.DBW 20;
      L     0;
      L     DB31.DBW 12;
      ==I;
      JC    M004;
      T     DB31.DBW 22;
      JU    M004;
M003: L     0;
      L     DB31.DBW 12;
      ==I;
      JC    M004;
      T     DB31.DBW 22;
M004: CLR;
END_FUNCTION

DATA_BLOCK DB 1
AUTHOR : FM
FAMILY : FM_CNT_1
NAME : CNT_CHAN
VERSION : 3.0
UDT 2
BEGIN
END_DATA_BLOCK

DATA_BLOCK DB 10
VERSION : 0.1
BEGIN
// 18 bytes; values not shown
END_DATA_BLOCK

DATA_BLOCK DB 11
VERSION : 0.1
BEGIN
// 18 bytes; values not shown
END_DATA_BLOCK

DATA_BLOCK DB 17
VERSION : 0.1
BEGIN
// 30 bytes; values not shown
END_DATA_BLOCK

DATA_BLOCK DB 18
VERSION : 0.1
BEGIN
// 30 bytes; values not shown
END_DATA_BLOCK

DATA_BLOCK DB 19
VERSION : 0.1
BEGIN
// 34 bytes; values not shown
END_DATA_BLOCK

DATA_BLOCK DB 20
VERSION : 0.1
BEGIN
// 34 bytes; values not shown
END_DATA_BLOCK

DATA_BLOCK DB 21
VERSION : 0.1
BEGIN
// 168 bytes; values not shown
END_DATA_BLOCK

DATA_BLOCK DB 22
VERSION : 0.1
BEGIN
// 66 bytes; values not shown
END_DATA_BLOCK

DATA_BLOCK DB 29
VERSION : 0.1
BEGIN
// 500 bytes; values not shown
END_DATA_BLOCK

DATA_BLOCK DB 30
VERSION : 0.1
BEGIN
// 74 bytes; values not shown
END_DATA_BLOCK

DATA_BLOCK DB 31
VERSION : 0.1
BEGIN
// 190 bytes; values not shown
END_DATA_BLOCK

DATA_BLOCK DB 32
VERSION : 0.1
BEGIN
// 48 bytes; values not shown
END_DATA_BLOCK

DATA_BLOCK DB 35
VERSION : 0.1
BEGIN
// 370 bytes; values not shown
END_DATA_BLOCK

DATA_BLOCK DB 39
VERSION : 0.1
BEGIN
// 500 bytes; values not shown
END_DATA_BLOCK

DATA_BLOCK DB 40
VERSION : 0.1
BEGIN
// 100 bytes; values not shown
END_DATA_BLOCK

DATA_BLOCK DB 41
VERSION : 0.1
BEGIN
// 102 bytes; values not shown
END_DATA_BLOCK

DATA_BLOCK DB 50
AUTHOR : SIMATIC
FAMILY : CP341
VERSION : 0.0
FB 8
BEGIN
END_DATA_BLOCK

DATA_BLOCK DB 51
AUTHOR : SIMATIC
FAMILY : CP341
VERSION : 0.0
FB 7
BEGIN
END_DATA_BLOCK

DATA_BLOCK DB 80
AUTHOR : SIMATIC
FAMILY : CP341
VERSION : 0.0
FB 7
BEGIN
END_DATA_BLOCK

DATA_BLOCK DB 100
VERSION : 0.1
BEGIN
// 222 bytes; values not shown
END_DATA_BLOCK

ORGANIZATION_BLOCK OB 1
VERSION : 0.1
BEGIN
// (block stored without names or comments; labels and parameter names are numbered)
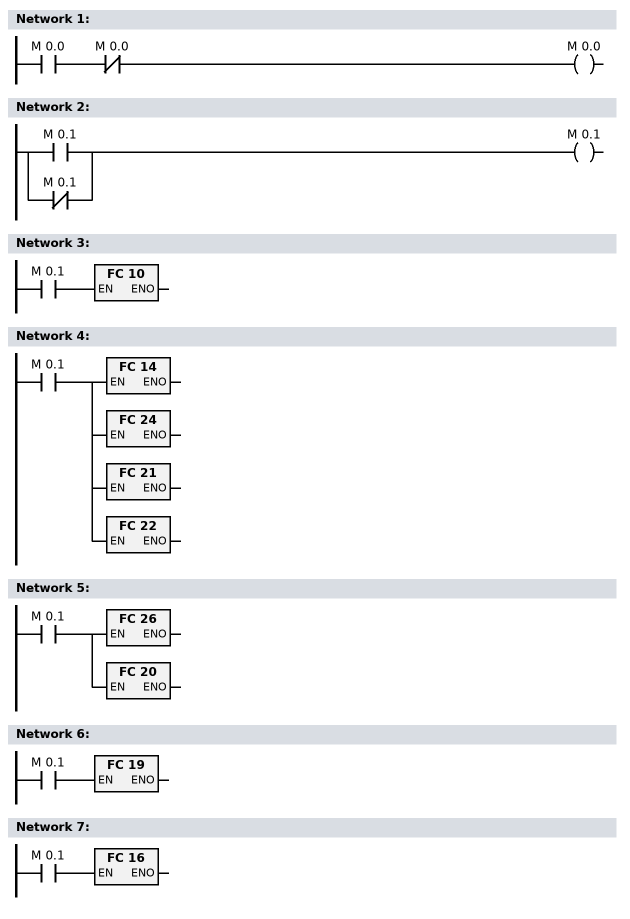
NETWORK
TITLE =
      A     M 0.0;
      AN    M 0.0;
      =     M 0.0;
NETWORK
TITLE =
      O     M 0.1;
      ON    M 0.1;
      =     M 0.1;
NETWORK
TITLE =
      A     M 0.1;
      JNB   M001;
      CALL  FC 10;
M001: NOP   0;
NETWORK
TITLE =
      A     M 0.1;
      =     L 20.0;
      A     L 20.0;
      JNB   M002;
      CALL  FC 14;
M002: NOP   0;
      A     L 20.0;
      JNB   M003;
      CALL  FC 24;
M003: NOP   0;
      A     L 20.0;
      JNB   M004;
      CALL  FC 21;
M004: NOP   0;
      A     L 20.0;
      JNB   M005;
      CALL  FC 22;
M005: NOP   0;
NETWORK
TITLE =
      A     M 0.1;
      =     L 20.0;
      A     L 20.0;
      JNB   M006;
      CALL  FC 26;
M006: NOP   0;
      A     L 20.0;
      JNB   M007;
      CALL  FC 20;
M007: NOP   0;
NETWORK
TITLE =
      A     M 0.1;
      JNB   M008;
      CALL  FC 19;
M008: NOP   0;
NETWORK
TITLE =
      A     M 0.1;
      JNB   M009;
      CALL  FC 16;
M009: NOP   0;
END_ORGANIZATION_BLOCK

ORGANIZATION_BLOCK OB 82
VERSION : 0.1
BEGIN
// (block stored without names or comments; labels and parameter names are numbered)
NETWORK
TITLE =
      SET;
      S     DB30.DBX 54.1;
      S     DB30.DBX 54.0;
      CALL  FC 4 (
           $1                       := 1,
           $2                       := DB30.DBW 72,
           $3                       := DB30.DBX 54.0);
END_ORGANIZATION_BLOCK

ORGANIZATION_BLOCK OB 86
VERSION : 0.1
BEGIN
// (block stored without names or comments; labels and parameter names are numbered)
NETWORK
TITLE =
END_ORGANIZATION_BLOCK

ORGANIZATION_BLOCK OB 100
VERSION : 0.1
BEGIN
// (block stored without names or comments; labels and parameter names are numbered)
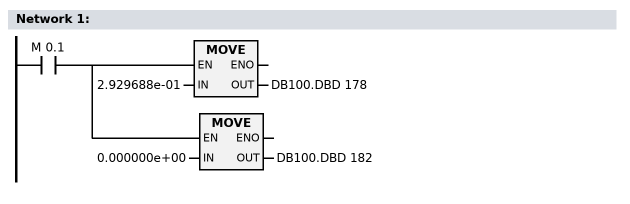
NETWORK
TITLE =
      A     M 0.1;
      =     L 20.0;
      A     L 20.0;
      JNB   M001;
      L     2.929688e-01;
      T     DB100.DBD 178;
M001: NOP   0;
      A     L 20.0;
      JNB   M002;
      L     0.000000e+00;
      T     DB100.DBD 182;
M002: NOP   0;
END_ORGANIZATION_BLOCK

ORGANIZATION_BLOCK OB 121
VERSION : 0.1
BEGIN
// (block stored without names or comments; labels and parameter names are numbered)
NETWORK
TITLE =
END_ORGANIZATION_BLOCK

ORGANIZATION_BLOCK OB 122
VERSION : 0.1
BEGIN
// (block stored without names or comments; labels and parameter names are numbered)
NETWORK
TITLE =
END_ORGANIZATION_BLOCK
